PROGRAM MAIN
VAR
	ntGetTime	: NT_GetTime;
	timeST		: Tc2_Utilities.TIMESTRUCT;
	
	ton			: TON;
	
	fbLocalSystemTime	: FB_LocalSystemTime;
END_VAR

ton(IN := NOT ton.Q, PT := T#100MS);

ntGetTime(
	NETID := '26.242.21.199.1.1',
	START := ton.Q,
	TIMESTR => timeST);
	
fbLocalSystemTime(
	sNetID:= '', 
	bEnable:= TRUE);

END_PROGRAM

(* stored: Version 1.1.0.1, ProductVersion 3.1.4024.5
   POU MAIN: Id {e8b40569-7154-4b82-b9cb-c910d5f73805}, SpecialFunc None *)
